Staubli VAL3: deleteItem.pgx

public program deleteItem(num& x_nIndex (dimensions=1))
  local num i
  local string l_sItem
begin
  // delete the selected item
  if pEditPoint.tData[x_nIndex].nType!=1 and size(pEditPoint.tData)>3
    // delete all the field
    delete(pEditPoint.tData[x_nIndex])
  else
    // not possible to delete the point
    if pEditPoint.tData[x_nIndex].nType!=1
      pEditPoint.tData[x_nIndex].pPoint.trsf={0,0,0,0,0,0}
    endIf
    x_nIndex=-1
  endIf
end
